ABB RobotStudio station: 6640_egm.rsstn

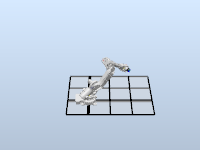
Station Station (saved by RobotStudio 21.4.9700.0)
Controller Controller_egm
  mechanical unit ROB_1: IRB6640_180_255__04, 6 joints, base frame (0, 0, 0) mm
Layout (positions relative to the parent item):
  - IRB6640_180_255__04 [mechanism, from Robots\IRB6640_180_255_G_04.rslib] at (0, 0, 0) mm; joint values [0.6276, 0.8397, -0.2375, 1.6757, -0.9007, 0.7954] (rad or m)
